(* IEC 61131-3 sources: AXOpen/src/showcase/app/src/components.kuka.robotics/Documentation, 7 files *)

(* ---- AxoKrc4_v_5_x_x_Krc5Showcase.st ---- *)
USING AXOpen.Core;

NAMESPACE AXOpen.Components.Kuka.Robotics
    {S7.extern=ReadWrite}
    CLASS AxoKrc4_v_5_x_x_Krc5Showcase EXTENDS AXOpen.Core.AxoObject
        //<ComponentDeclaration>
        VAR PUBLIC
            // KRC5 controller driven by the same AxoKrc4 proxy —
            // the slot-2 DIO512 layout is identical between KRC4 and KRC5.
            ExampleRobot : AXOpen.Components.Kuka.Robotics.v_5_x_x.AxoKrc4;
        END_VAR
        //</ComponentDeclaration>

        //<InitializationArgumentsDeclaration>
        VAR PUBLIC
            movementParams : AXOpen.Components.Abstractions.Robotics.AxoRoboticsMovementsParams;
            {#ix-set:AttributeName = "<#Activate manual control#>"}
            ActivateManualControl : BOOL;
        END_VAR
        //</InitializationArgumentsDeclaration>

        METHOD PUBLIC OVERRIDE Run
            VAR_INPUT
                inParent : IAxoObject;
            END_VAR

            SUPER.Run(inParent);

            IF ActivateManualControl THEN
                ExampleRobot.ActivateManualControl();
            END_IF;

            //<Initialization>
            // kuka_rb2_HwID points at the KRC5 device (192.168.100.106)
            // provisioned by the kuka_krc5_dio512 template in plc_line.hwl.yml.
            ExampleRobot.Run(THIS, AXOpen.Showcase.HwIdentifiers#kuka_rb2_HwID);
            //</Initialization>

            THIS.UseInSequencer();
        END_METHOD

        //<Usage>
        VAR PUBLIC
            Sequencer : AxoSequencer;
            Steps : ARRAY[0..19] OF AXOpen.Core.AxoStep;
        END_VAR

        METHOD PRIVATE UseInSequencer

            Sequencer.Run(THIS);
            Sequencer.Open();
            Sequencer.SequenceMode := eAxoSequenceMode#RunOnce;

            IF(Steps[0].Execute(Sequencer, 'Restore')) THEN
                ActivateManualControl := FALSE;
                ExampleRobot.Config.InfoTime      := LTIME#2S;
                ExampleRobot.Config.TaskTimeout   := LTIME#0S;
                ExampleRobot.Config.ErrorTime     := LTIME#0S;
                ExampleRobot.Restore();
                Sequencer.MoveNext();
            END_IF;

            IF(Steps[1].Execute(Sequencer, 'Start at main')) THEN
                IF(ExampleRobot.StartAtMain().IsDone()) THEN
                    Sequencer.MoveNext();
                END_IF;
            END_IF;

            IF(Steps[2].Execute(Sequencer, 'Start motors and program')) THEN
                IF(ExampleRobot.StartMotorsAndProgram().IsDone()) THEN
                    Sequencer.MoveNext();
                END_IF;
            END_IF;

            IF(Steps[3].Execute(Sequencer, 'Move to position 100')) THEN
                movementParams.ActionNo         :=  BYTE#100;
                movementParams.GlobalSpeed      :=  BYTE#5;
                movementParams.ToolNo           :=  BYTE#10;
                movementParams.WorkobjectNo     :=  BYTE#15;
                movementParams.PointNo          :=  BYTE#20;
                movementParams.UserSpecSpeed1   :=  INT#25;
                movementParams.UserSpecSpeed2   :=  INT#30;
                movementParams.Coordinates.X    :=  REAL#-1.2;
                movementParams.Coordinates.Y    :=  REAL#2.3;
                movementParams.Coordinates.Z    :=  REAL#3.4;
                movementParams.Coordinates.Rx   :=  REAL#4.5;
                movementParams.Coordinates.Ry   :=  REAL#5.6;
                movementParams.Coordinates.Rz   :=  REAL#6.7;

                IF(ExampleRobot.StartMovements(movementParams).IsDone()) THEN
                    ExampleRobot.StartMovementsTask.Restore();
                    Sequencer.MoveNext();
                END_IF;
            END_IF;

            IF(Steps[4].Execute(Sequencer, 'Move to position 1')) THEN
                movementParams.ActionNo             :=  BYTE#1;

                IF(ExampleRobot.StartMovements(movementParams).IsDone()) THEN
                    ExampleRobot.StartMovementsTask.Restore();
                    Sequencer.MoveNext();
                END_IF;
            END_IF;

            IF(Steps[5].Execute(Sequencer, 'Move to position 3')) THEN
                movementParams.ActionNo             :=  BYTE#3;

                IF(ExampleRobot.StartMovements(movementParams).IsBusy() AND Sequencer.CurrentStep.Duration >= T#500ms) THEN
                    Sequencer.MoveNext();
                END_IF;
            END_IF;

            IF(Steps[6].Execute(Sequencer, 'Stop during movement')) THEN
                ExampleRobot.StartMovements(movementParams);
                IF(ExampleRobot.StopMovements().IsDone()) THEN
                    Sequencer.MoveNext();
                END_IF;
            END_IF;

            IF(Steps[7].Execute(Sequencer, '<#Unlocking and opening the robotic cell#>')) THEN
                ExampleRobot.StartMovements(movementParams);
                IF (Sequencer.CurrentStep.Duration >= T#1s) THEN
                    Sequencer.MoveNext();
                END_IF;
            END_IF;

            IF (Steps[8].Execute(Sequencer, '<#Closing and locking the robotic cell#>')) THEN
                ExampleRobot.StartMovements(movementParams);
                IF (Sequencer.CurrentStep.Duration >= T#1s) THEN
                    Sequencer.MoveNext();
                END_IF;
            END_IF;

            IF(Steps[9].Execute(Sequencer, 'Start motors and program')) THEN
                ExampleRobot.StartMovements(movementParams);
                IF(ExampleRobot.StartMotorsAndProgram().IsDone() AND Sequencer.CurrentStep.Duration >= T#1s) THEN
                    Sequencer.MoveNext();
                END_IF;
            END_IF;

            IF(Steps[10].Execute(Sequencer, 'Continue to position 3')) THEN
                ExampleRobot.StartMovements(movementParams);
                IF(ExampleRobot.StartMovementsTask.IsDone()) THEN
                    ExampleRobot.StartMovementsTask.Restore();
                    Sequencer.MoveNext();
                END_IF;
            END_IF;

            IF(Steps[11].Execute(Sequencer, 'Move to position 100')) THEN
                movementParams.ActionNo             :=  BYTE#100;

                IF(ExampleRobot.StartMovements(movementParams).IsDone()) THEN
                    ExampleRobot.StartMovementsTask.Restore();
                    Sequencer.MoveNext();
                END_IF;
            END_IF;

            IF(Steps[12].Execute(Sequencer, 'Move to position 1')) THEN
                movementParams.ActionNo             :=  BYTE#1;

                IF(ExampleRobot.StartMovements(movementParams).IsDone()) THEN
                    ExampleRobot.StartMovementsTask.Restore();
                    Sequencer.MoveNext();
                END_IF;
            END_IF;

            IF(Steps[13].Execute(Sequencer, 'Stop movement and program')) THEN
                IF(ExampleRobot.StopMovementsAndProgram().IsDone()) THEN
                    Sequencer.MoveNext();
                END_IF;
            END_IF;

            IF(Steps[14].Execute(Sequencer, 'Stop motors')) THEN
                IF(ExampleRobot.StopMotors().IsDone()) THEN
                    Sequencer.MoveNext();
                END_IF;
            END_IF;

            IF(Steps[15].Execute(Sequencer, 'Reset all outputs')) THEN
                IF(ExampleRobot.ResetAllOutputs().IsDone()) THEN
                    Sequencer.MoveNext();
                END_IF;
            END_IF;

            IF(Steps[16].Execute(Sequencer, 'Start motors, program and movements combined')) THEN
                IF(ExampleRobot.StartMotorsProgramAndMovements(movementParams).IsDone()) THEN
                    Sequencer.MoveNext();
                END_IF;
            END_IF;

            IF(Steps[17].Execute(Sequencer, 'Stop program')) THEN
                IF(ExampleRobot.StopProgram().IsDone()) THEN
                    Sequencer.MoveNext();
                END_IF;
            END_IF;

            IF(Steps[18].Execute(Sequencer, 'Start program')) THEN
                IF(ExampleRobot.StartProgram().IsDone()) THEN
                    Sequencer.MoveNext();
                END_IF;
            END_IF;

            IF(Steps[19].Execute(Sequencer, 'Restore')) THEN
                ExampleRobot.Restore();
                Sequencer.CompleteSequence();
            END_IF;
        END_METHOD

        //</Usage>
    END_CLASS
END_NAMESPACE

(* ---- AxoKrc4_v_5_x_x_ManualControl.st ---- *)
USING AXOpen.Core;
USING AXOpen.Components.Abstractions.Robotics;

NAMESPACE AXOpen.Components.Kuka.Robotics.v_5_x_x
    {S7.extern=ReadWrite}
    CLASS AxoKrc4_v_5_x_x_ManualControl EXTENDS AXOpen.Core.AxoObject
        //<ComponentDeclaration>
        VAR PUBLIC
            ManualRobot : AXOpen.Components.Kuka.Robotics.v_5_x_x.AxoKrc4;
        END_VAR
        //</ComponentDeclaration>

        //<InitializationArgumentsDeclaration>
        VAR PUBLIC
            manualMovementParams : AXOpen.Components.Abstractions.Robotics.AxoRoboticsMovementsParams;
            {#ix-set:AttributeName = "<#Engage manual control#>"}
            EngageManualControl : BOOL;
            {#ix-set:AttributeName = "<#Trigger manual move (one shot)#>"}
            TriggerManualMove : BOOL;
        END_VAR
        //</InitializationArgumentsDeclaration>

        METHOD PUBLIC OVERRIDE Run
            VAR_INPUT
                inParent : IAxoObject;
            END_VAR

            SUPER.Run(inParent);

            ManualRobot.Config.InfoTime    := LTIME#2S;
            ManualRobot.Config.ErrorTime   := LTIME#0S;
            ManualRobot.Config.TaskTimeout := LTIME#0S;

            //<Initialization>
            ManualRobot.Run(inParent := THIS,
                            hwID     := AXOpen.Showcase.HwIdentifiers#kuka_rb1_HwID);
            //</Initialization>

            //<ManualControlActivation>
            // ActivateManualControl() must be called every cycle while the
            // operator drives the component from the HMI. The component
            // bypasses the automatic task pipeline and exposes raw command
            // signals through its dedicated views.
            IF EngageManualControl THEN
                ManualRobot.ActivateManualControl();
            END_IF;
            //</ManualControlActivation>

            //<ManualMoveTrigger>
            // The HMI can pre-load movement parameters and fire a single
            // StartMovements() invocation. When the task completes the
            // operator restores it from its terminal state to be ready
            // for the next manual command.
            IF TriggerManualMove THEN
                manualMovementParams.ActionNo       :=  BYTE#1;
                manualMovementParams.GlobalSpeed    :=  BYTE#10;
                manualMovementParams.ToolNo         :=  BYTE#1;
                manualMovementParams.WorkobjectNo   :=  BYTE#1;
                manualMovementParams.PointNo        :=  BYTE#1;
                IF ManualRobot.StartMovements(manualMovementParams).IsDone() THEN
                    ManualRobot.StartMovementsTask.Restore();
                    TriggerManualMove := FALSE;
                END_IF;
            END_IF;
            //</ManualMoveTrigger>
        END_METHOD
    END_CLASS
END_NAMESPACE

(* ---- AxoKrc4_v_5_x_x_Showcase.st ---- *)
USING AXOpen.Core;
USING AXOpen.Components.Abstractions.Robotics;

NAMESPACE AXOpen.Components.Kuka.Robotics.v_5_x_x
    {S7.extern=ReadWrite}
    CLASS AxoKrc4_v_5_x_x_Showcase EXTENDS AXOpen.Core.AxoObject
        //<ComponentDeclaration>
        VAR PUBLIC
            ExampleRobot : AXOpen.Components.Kuka.Robotics.v_5_x_x.AxoKrc4;
        END_VAR
        //</ComponentDeclaration>

        //<InitializationArgumentsDeclaration>
        VAR PUBLIC
            movementParams : AXOpen.Components.Abstractions.Robotics.AxoRoboticsMovementsParams;
            {#ix-set:AttributeName = "<#Activate manual control#>"}
            ActivateManualControl : BOOL;
        END_VAR
        //</InitializationArgumentsDeclaration>

        METHOD PUBLIC OVERRIDE Run
            VAR_INPUT
                inParent : IAxoObject;
            END_VAR

            SUPER.Run(inParent);

            IF ActivateManualControl THEN
                ExampleRobot.ActivateManualControl();
            END_IF;

            ExampleRobot.Config.ErrorTime := T#0s;
            //<Initialization>
            ExampleRobot.Run(THIS,AXOpen.Showcase.HwIdentifiers#kuka_rb1_HwID);
            //</Initialization>

        THIS.UseInSequencer();
        END_METHOD

        //<Usage>
        VAR PUBLIC
            Sequencer : AxoSequencer;
            Steps : ARRAY[0..19] OF AXOpen.Core.AxoStep;
        END_VAR

        METHOD PRIVATE UseInSequencer

            Sequencer.Run(THIS);
            Sequencer.Open();
            Sequencer.SequenceMode := eAxoSequenceMode#RunOnce;

            IF(Steps[0].Execute(Sequencer, 'Restore')) THEN
                ActivateManualControl := FALSE;
                ExampleRobot.Config.InfoTime      := LTIME#2S;
                ExampleRobot.Config.TaskTimeout   := LTIME#0S;
                ExampleRobot.Config.ErrorTime     := LTIME#0S;
                ExampleRobot.Restore();
                Sequencer.MoveNext();
            END_IF;

            IF(Steps[1].Execute(Sequencer, 'Start at main')) THEN
                IF(ExampleRobot.StartAtMain().IsDone()) THEN
                    Sequencer.MoveNext();
                END_IF;
            END_IF;

            IF(Steps[2].Execute(Sequencer, 'Start motors and program')) THEN
                IF(ExampleRobot.StartMotorsAndProgram().IsDone()) THEN
                    Sequencer.MoveNext();
                END_IF;
            END_IF;

            IF(Steps[3].Execute(Sequencer, 'Move to position 100')) THEN
                movementParams.ActionNo         :=  BYTE#100;
                movementParams.GlobalSpeed      :=  BYTE#5;
                movementParams.ToolNo           :=  BYTE#10;
                movementParams.WorkobjectNo     :=  BYTE#15;
                movementParams.PointNo          :=  BYTE#20;
                movementParams.UserSpecSpeed1   :=  INT#25;
                movementParams.UserSpecSpeed2   :=  INT#30;
                movementParams.Coordinates.X    :=  REAL#-1.2;
                movementParams.Coordinates.Y    :=  REAL#2.3;
                movementParams.Coordinates.Z    :=  REAL#3.4;
                movementParams.Coordinates.Rx   :=  REAL#4.5;
                movementParams.Coordinates.Ry   :=  REAL#5.6;
                movementParams.Coordinates.Rz   :=  REAL#6.7;

                IF(ExampleRobot.StartMovements(movementParams).IsDone()) THEN
                    ExampleRobot.StartMovementsTask.Restore();
                    Sequencer.MoveNext();
                END_IF;
            END_IF;

            IF(Steps[4].Execute(Sequencer, 'Move to position 1')) THEN
                movementParams.ActionNo             :=  BYTE#1;

                IF(ExampleRobot.StartMovements(movementParams).IsDone()) THEN
                    ExampleRobot.StartMovementsTask.Restore();
                    Sequencer.MoveNext();
                END_IF;
            END_IF;

            IF(Steps[5].Execute(Sequencer, 'Move to position 3')) THEN
                movementParams.ActionNo             :=  BYTE#3;

                IF(ExampleRobot.StartMovements(movementParams).IsBusy() AND Sequencer.CurrentStep.Duration >= T#500ms) THEN
                    Sequencer.MoveNext();
                END_IF;
            END_IF;
            // Simulation of the entering the robotic cell during movement =>
            IF(Steps[6].Execute(Sequencer, 'Stop during movement')) THEN
                ExampleRobot.StartMovements(movementParams); // <- This line just emulates the cyclical call of the movement method
                IF(ExampleRobot.StopMovements(eAxoRoboticsStopType#Soft).IsDone()) THEN
                    Sequencer.MoveNext();
                END_IF;
            END_IF;

            IF(Steps[7].Execute(Sequencer, '<#Unlocking and opening the robotic cell#>')) THEN
                //-------------------------------------------------------
                ExampleRobot.StartMovements(movementParams); // <- This line just emulates the cyclical call of the movement method
                IF (Sequencer.CurrentStep.Duration >= T#1s) THEN    // IF (TRUE) THEN
                    Sequencer.MoveNext();
                END_IF;
                //-------------------------------------------------------
            END_IF;

            IF (Steps[8].Execute(Sequencer, '<#Closing and locking the robotic cell#>')) THEN
                //-------------------------------------------------------
                ExampleRobot.StartMovements(movementParams); // <- This line just emulates the cyclical call of the movement method
                IF (Sequencer.CurrentStep.Duration >= T#1s) THEN    // IF (TRUE) THEN
                    Sequencer.MoveNext();
                END_IF;
                //-------------------------------------------------------
            END_IF;
            // <= Simulation of the entering the robotic cell during movement

            IF(Steps[9].Execute(Sequencer, 'Start motors and program')) THEN
                ExampleRobot.StartMovements(movementParams); // <- This line just emulates the cyclical call of the movement method
                IF(ExampleRobot.StartMotorsAndProgram().IsDone() AND Sequencer.CurrentStep.Duration >= T#1s) THEN //IF(ExampleRobot.StartMotorsAndProgram().IsDone()) THEN // <- Starting motor and program after safety circuit has been interupted
                    Sequencer.MoveNext();
                END_IF;
            END_IF;

            IF(Steps[10].Execute(Sequencer, 'Continue to position 3')) THEN
                ExampleRobot.StartMovements(movementParams); // <- This line just emulates the cyclical call of the movement method
                IF(ExampleRobot.StartMovementsTask.IsDone()) THEN
                    ExampleRobot.StartMovementsTask.Restore();
                    Sequencer.MoveNext();
                END_IF;
            END_IF;

            IF(Steps[11].Execute(Sequencer, 'Move to position 100')) THEN
                movementParams.ActionNo             :=  BYTE#100;

                IF(ExampleRobot.StartMovements(movementParams).IsDone()) THEN
                    ExampleRobot.StartMovementsTask.Restore();
                    Sequencer.MoveNext();
                END_IF;
            END_IF;

            IF(Steps[12].Execute(Sequencer, 'Move to position 1')) THEN
                movementParams.ActionNo             :=  BYTE#1;

                IF(ExampleRobot.StartMovements(movementParams).IsDone()) THEN
                    ExampleRobot.StartMovementsTask.Restore();
                    Sequencer.MoveNext();
                END_IF;
            END_IF;

            IF(Steps[13].Execute(Sequencer, 'Stop movement and program')) THEN
                IF(ExampleRobot.StopMovementsAndProgram(eAxoRoboticsStopType#Soft).IsDone()) THEN
                    Sequencer.MoveNext();
                END_IF;
            END_IF;

            IF(Steps[14].Execute(Sequencer, 'Stop motors')) THEN
                IF(ExampleRobot.StopMotors().IsDone()) THEN
                    Sequencer.MoveNext();
                END_IF;
            END_IF;

            IF(Steps[15].Execute(Sequencer, 'Reset all outputs')) THEN
                IF(ExampleRobot.ResetAllOutputs().IsDone()) THEN
                    Sequencer.MoveNext();
                END_IF;
            END_IF;

            IF(Steps[16].Execute(Sequencer, 'Start motors, program and movements combined')) THEN
                IF(ExampleRobot.StartMotorsProgramAndMovements(movementParams).IsDone()) THEN
                    Sequencer.MoveNext();
                END_IF;
            END_IF;

            IF(Steps[17].Execute(Sequencer, 'Stop program')) THEN
                IF(ExampleRobot.StopProgram().IsDone()) THEN
                    Sequencer.MoveNext();
                END_IF;
            END_IF;

            IF(Steps[18].Execute(Sequencer, 'Start program')) THEN
                IF(ExampleRobot.StartProgram().IsDone()) THEN
                    Sequencer.MoveNext();
                END_IF;
            END_IF;

            IF(Steps[19].Execute(Sequencer, 'Restore')) THEN
                ExampleRobot.Restore();
                Sequencer.CompleteSequence();
            END_IF;
        END_METHOD

        //</Usage>
    END_CLASS
END_NAMESPACE

(* ---- AxoKrc4_v_5_x_x_Showcase2.st ---- *)
USING AXOpen.Core;

NAMESPACE AXOpen.Components.Kuka.Robotics
    {S7.extern=ReadWrite}
    CLASS AxoKrc4_v_5_x_x_Showcase2 EXTENDS AXOpen.Core.AxoObject
        //<ComponentDeclaration>
        VAR PUBLIC
            ExampleRobot : AXOpen.Components.Kuka.Robotics.v_5_x_x.AxoKrc4;
        END_VAR
        //</ComponentDeclaration>

        //<InitializationArgumentsDeclaration>
        VAR PUBLIC
            movementParams : AXOpen.Components.Abstractions.Robotics.AxoRoboticsMovementsParams;
            {#ix-set:AttributeName = "<#Activate manual control#>"}
            ActivateManualControl : BOOL;
        END_VAR
        //</InitializationArgumentsDeclaration>

        METHOD PUBLIC OVERRIDE Run
            VAR_INPUT
                inParent : IAxoObject;
            END_VAR

            SUPER.Run(inParent);

            IF ActivateManualControl THEN
                ExampleRobot.ActivateManualControl();
            END_IF;

            //<Initialization>
            ExampleRobot.Run(THIS,AXOpen.Showcase.HwIdentifiers#kuka_rb1_HwID);
            //</Initialization>

            THIS.UseInSequencer();
        END_METHOD

        //<Usage>
        VAR PUBLIC
            Sequencer : AxoSequencer;
            Steps : ARRAY[0..14] OF AXOpen.Core.AxoStep;
        END_VAR

        METHOD PRIVATE UseInSequencer

            Sequencer.Run(THIS);
            Sequencer.Open();
            Sequencer.SequenceMode := eAxoSequenceMode#RunOnce;

            IF(Steps[0].Execute(Sequencer, 'Restore')) THEN
                ActivateManualControl := FALSE;
                ExampleRobot.Config.TaskTimeout   := LTIME#0S;
                ExampleRobot.Config.ErrorTime     := LTIME#0S;
                ExampleRobot.Restore();
                Sequencer.MoveNext();
            END_IF;

            IF(Steps[1].Execute(Sequencer, 'Start at main')) THEN
                IF(ExampleRobot.StartAtMain().IsDone()) THEN
                    Sequencer.MoveNext();
                END_IF;
            END_IF;

            IF(Steps[2].Execute(Sequencer, 'Start motors and program')) THEN
                IF(ExampleRobot.StartMotorsAndProgram().IsDone()) THEN
                    Sequencer.MoveNext();
                END_IF;
            END_IF;

            IF(Steps[3].Execute(Sequencer, 'Move to position 100')) THEN
                movementParams.ActionNo         :=  BYTE#100;
                movementParams.GlobalSpeed      :=  BYTE#5;
                movementParams.ToolNo           :=  BYTE#10;
                movementParams.WorkobjectNo     :=  BYTE#15;
                movementParams.PointNo          :=  BYTE#20;
                movementParams.UserSpecSpeed1   :=  INT#25;
                movementParams.UserSpecSpeed2   :=  INT#30;
                movementParams.Coordinates.X    :=  REAL#-1.2;
                movementParams.Coordinates.Y    :=  REAL#2.3;
                movementParams.Coordinates.Z    :=  REAL#3.4;
                movementParams.Coordinates.Rx   :=  REAL#4.5;
                movementParams.Coordinates.Ry   :=  REAL#5.6;
                movementParams.Coordinates.Rz   :=  REAL#6.7;

                IF(ExampleRobot.StartMovements(movementParams).IsDone()) THEN
                    ExampleRobot.StartMovementsTask.Restore();
                    Sequencer.MoveNext();
                END_IF;
            END_IF;

            IF(Steps[4].Execute(Sequencer, 'Move to position 1')) THEN
                movementParams.ActionNo             :=  BYTE#1;

                IF(ExampleRobot.StartMovements(movementParams).IsDone()) THEN
                    ExampleRobot.StartMovementsTask.Restore();
                    Sequencer.MoveNext();
                END_IF;
            END_IF;

            IF(Steps[5].Execute(Sequencer, 'Move to position 3')) THEN
                movementParams.ActionNo             :=  BYTE#3;

                IF(ExampleRobot.StartMovements(movementParams).IsBusy() AND Sequencer.CurrentStep.Duration >= T#500ms) THEN
                    Sequencer.MoveNext();
                END_IF;
            END_IF;
            // Simulation of the entering the robotic cell during movement =>
            IF(Steps[6].Execute(Sequencer, 'Stop during movement')) THEN
                ExampleRobot.StartMovements(movementParams); // <- This line just emulates the cyclical call of the movement method
                IF(ExampleRobot.StopMovements().IsDone()) THEN
                    Sequencer.MoveNext();
                END_IF;
            END_IF;

            IF(Steps[7].Execute(Sequencer, '<#Unlocking and opening the robotic cell#>')) THEN
                //-------------------------------------------------------
                ExampleRobot.StartMovements(movementParams); // <- This line just emulates the cyclical call of the movement method
                IF (Sequencer.CurrentStep.Duration >= T#1s) THEN    // IF (TRUE) THEN
                    Sequencer.MoveNext();
                END_IF;
                //-------------------------------------------------------
            END_IF;

            IF (Steps[8].Execute(Sequencer, '<#Closing and locking the robotic cell#>')) THEN
                //-------------------------------------------------------
                ExampleRobot.StartMovements(movementParams); // <- This line just emulates the cyclical call of the movement method
                IF (Sequencer.CurrentStep.Duration >= T#1s) THEN    // IF (TRUE) THEN
                    Sequencer.MoveNext();
                END_IF;
                //-------------------------------------------------------
            END_IF;
            // <= Simulation of the entering the robotic cell during movement

            IF(Steps[9].Execute(Sequencer, 'Start motors and program')) THEN
                ExampleRobot.StartMovements(movementParams); // <- This line just emulates the cyclical call of the movement method
                IF(ExampleRobot.StartMotorsAndProgram().IsDone() AND Sequencer.CurrentStep.Duration >= T#1s) THEN //IF(ExampleRobot.StartMotorsAndProgram().IsDone()) THEN // <- Starting motor and program after safety circuit has been interupted
                    Sequencer.MoveNext();
                END_IF;
            END_IF;

            IF(Steps[10].Execute(Sequencer, 'Continue to position 3')) THEN
                ExampleRobot.StartMovements(movementParams); // <- This line just emulates the cyclical call of the movement method
                IF(ExampleRobot.StartMovementsTask.IsDone()) THEN
                    ExampleRobot.StartMovementsTask.Restore();
                    Sequencer.MoveNext();
                END_IF;
            END_IF;

            IF(Steps[11].Execute(Sequencer, 'Move to position 100')) THEN
                movementParams.ActionNo             :=  BYTE#100;

                IF(ExampleRobot.StartMovements(movementParams).IsDone()) THEN
                    ExampleRobot.StartMovementsTask.Restore();
                    Sequencer.MoveNext();
                END_IF;
            END_IF;

            IF(Steps[12].Execute(Sequencer, 'Move to position 1')) THEN
                movementParams.ActionNo             :=  BYTE#1;

                IF(ExampleRobot.StartMovements(movementParams).IsDone()) THEN
                    ExampleRobot.StartMovementsTask.Restore();
                    Sequencer.MoveNext();
                END_IF;
            END_IF;

            IF(Steps[13].Execute(Sequencer, 'Stop movement and program')) THEN
                IF(ExampleRobot.StopMovementsAndProgram().IsDone()) THEN
                    Sequencer.MoveNext();
                END_IF;
            END_IF;
            IF(Steps[14].Execute(Sequencer, 'Restore')) THEN
                ExampleRobot.Restore();
                Sequencer.CompleteSequence();
            END_IF;
        END_METHOD

        //</Usage>
    END_CLASS
END_NAMESPACE

(* ---- AxoKrc5_v_5_x_x_ManualControl.st ---- *)
USING AXOpen.Core;
USING AXOpen.Components.Abstractions.Robotics;

NAMESPACE AXOpen.Components.Kuka.Robotics.v_5_x_x
    {S7.extern=ReadWrite}
    CLASS AxoKrc5_v_5_x_x_ManualControl EXTENDS AXOpen.Core.AxoObject
        //<ComponentDeclaration>
        VAR PUBLIC
            ManualRobot : AXOpen.Components.Kuka.Robotics.v_5_x_x.AxoKrc5;
        END_VAR
        //</ComponentDeclaration>

        //<InitializationArgumentsDeclaration>
        VAR PUBLIC
            manualMovementParams : AXOpen.Components.Abstractions.Robotics.AxoRoboticsMovementsParams;
            {#ix-set:AttributeName = "<#Engage manual control#>"}
            EngageManualControl : BOOL;
            {#ix-set:AttributeName = "<#Trigger manual move (one shot)#>"}
            TriggerManualMove : BOOL;
        END_VAR
        //</InitializationArgumentsDeclaration>

        METHOD PUBLIC OVERRIDE Run
            VAR_INPUT
                inParent : IAxoObject;
            END_VAR

            SUPER.Run(inParent);

            ManualRobot.Config.InfoTime    := LTIME#2S;
            ManualRobot.Config.ErrorTime   := LTIME#0S;
            ManualRobot.Config.TaskTimeout := LTIME#0S;

            //<Initialization>
            ManualRobot.Run(inParent := THIS,
                            hwID     := AXOpen.Showcase.HwIdentifiers#kuka_rb2_HwID);
            //</Initialization>

            //<ManualControlActivation>
            // ActivateManualControl() must be called every cycle while the
            // operator drives the component from the HMI. The component
            // bypasses the automatic task pipeline and exposes raw command
            // signals through its dedicated views.
            IF EngageManualControl THEN
                ManualRobot.ActivateManualControl();
            END_IF;
            //</ManualControlActivation>

            //<ManualMoveTrigger>
            // The HMI can pre-load movement parameters and fire a single
            // StartMovements() invocation. When the task completes the
            // operator restores it from its terminal state to be ready
            // for the next manual command.
            IF TriggerManualMove THEN
                manualMovementParams.ActionNo       :=  BYTE#1;
                manualMovementParams.GlobalSpeed    :=  BYTE#10;
                manualMovementParams.ToolNo         :=  BYTE#1;
                manualMovementParams.WorkobjectNo   :=  BYTE#1;
                manualMovementParams.PointNo        :=  BYTE#1;
                IF ManualRobot.StartMovements(manualMovementParams).IsDone() THEN
                    ManualRobot.StartMovementsTask.Restore();
                    TriggerManualMove := FALSE;
                END_IF;
            END_IF;
            //</ManualMoveTrigger>
        END_METHOD
    END_CLASS
END_NAMESPACE

(* ---- AxoKrc5_v_5_x_x_Showcase.st ---- *)
USING AXOpen.Core;
USING AXOpen.Components.Abstractions.Robotics;

NAMESPACE AXOpen.Components.Kuka.Robotics.v_5_x_x
    {S7.extern=ReadWrite}
    CLASS AxoKrc5_v_5_x_x_Showcase EXTENDS AXOpen.Core.AxoObject
        //<ComponentDeclaration>
        VAR PUBLIC
            ExampleRobot : AXOpen.Components.Kuka.Robotics.v_5_x_x.AxoKrc5;
        END_VAR
        //</ComponentDeclaration>

        //<InitializationArgumentsDeclaration>
        VAR PUBLIC
            movementParams : AXOpen.Components.Abstractions.Robotics.AxoRoboticsMovementsParams;
            {#ix-set:AttributeName = "<#Activate manual control#>"}
            ActivateManualControl : BOOL;
        END_VAR
        //</InitializationArgumentsDeclaration>

        METHOD PUBLIC OVERRIDE Run
            VAR_INPUT
                inParent : IAxoObject;
            END_VAR

            SUPER.Run(inParent);

            IF ActivateManualControl THEN
                ExampleRobot.ActivateManualControl();
            END_IF;

            //<Initialization>
            ExampleRobot.Run(THIS,AXOpen.Showcase.HwIdentifiers#kuka_rb2_HwID);
            //</Initialization>

            THIS.UseInSequencer();
        END_METHOD

        //<Usage>
        VAR PUBLIC
            Sequencer : AxoSequencer;
            Steps : ARRAY[0..20] OF AXOpen.Core.AxoStep;
            {#ix-set:AttributeName = "<#Last byte received from robot#>"}
            _lastByteFromRobot : BYTE;
        END_VAR

        METHOD PRIVATE UseInSequencer

            Sequencer.Run(THIS);
            Sequencer.Open();
            Sequencer.SequenceMode := eAxoSequenceMode#RunOnce;

            IF(Steps[0].Execute(Sequencer, 'Restore')) THEN
                ActivateManualControl := FALSE;
                ExampleRobot.Config.InfoTime      := LTIME#2S;
                ExampleRobot.Config.TaskTimeout   := LTIME#0S;
                ExampleRobot.Config.ErrorTime     := LTIME#0S;
                ExampleRobot.Restore();
                Sequencer.MoveNext();
            END_IF;

            IF(Steps[1].Execute(Sequencer, 'Start at main')) THEN
                IF(ExampleRobot.StartAtMain().IsDone()) THEN
                    Sequencer.MoveNext();
                END_IF;
            END_IF;

            IF(Steps[2].Execute(Sequencer, 'Start motors and program')) THEN
                IF(ExampleRobot.StartMotorsAndProgram().IsDone()) THEN
                    Sequencer.MoveNext();
                END_IF;
            END_IF;

            IF(Steps[3].Execute(Sequencer, 'Move to position 100')) THEN
                movementParams.ActionNo         :=  BYTE#100;
                movementParams.GlobalSpeed      :=  BYTE#5;
                movementParams.ToolNo           :=  BYTE#10;
                movementParams.WorkobjectNo     :=  BYTE#15;
                movementParams.PointNo          :=  BYTE#20;
                movementParams.UserSpecSpeed1   :=  INT#25;
                movementParams.UserSpecSpeed2   :=  INT#30;
                movementParams.Coordinates.X    :=  REAL#-1.2;
                movementParams.Coordinates.Y    :=  REAL#2.3;
                movementParams.Coordinates.Z    :=  REAL#3.4;
                movementParams.Coordinates.Rx   :=  REAL#4.5;
                movementParams.Coordinates.Ry   :=  REAL#5.6;
                movementParams.Coordinates.Rz   :=  REAL#6.7;

                IF(ExampleRobot.StartMovements(movementParams).IsDone()) THEN
                    ExampleRobot.StartMovementsTask.Restore();
                    Sequencer.MoveNext();
                END_IF;
            END_IF;

            IF(Steps[4].Execute(Sequencer, 'Move to position 1')) THEN
                movementParams.ActionNo             :=  BYTE#1;

                IF(ExampleRobot.StartMovements(movementParams).IsDone()) THEN
                    ExampleRobot.StartMovementsTask.Restore();
                    Sequencer.MoveNext();
                END_IF;
            END_IF;

            IF(Steps[5].Execute(Sequencer, 'Move to position 3')) THEN
                movementParams.ActionNo             :=  BYTE#3;

                IF(ExampleRobot.StartMovements(movementParams).IsBusy() AND Sequencer.CurrentStep.Duration >= T#500ms) THEN
                    Sequencer.MoveNext();
                END_IF;
            END_IF;
            // Simulation of the entering the robotic cell during movement =>
            IF(Steps[6].Execute(Sequencer, 'Stop during movement')) THEN
                ExampleRobot.StartMovements(movementParams); // <- This line just emulates the cyclical call of the movement method
                IF(ExampleRobot.StopMovements(eAxoRoboticsStopType#Soft).IsDone()) THEN
                    Sequencer.MoveNext();
                END_IF;
            END_IF;

            IF(Steps[7].Execute(Sequencer, '<#Unlocking and opening the robotic cell#>')) THEN
                //-------------------------------------------------------
                ExampleRobot.StartMovements(movementParams); // <- This line just emulates the cyclical call of the movement method
                IF (Sequencer.CurrentStep.Duration >= T#1s) THEN    // IF (TRUE) THEN
                    Sequencer.MoveNext();
                END_IF;
                //-------------------------------------------------------
            END_IF;

            IF (Steps[8].Execute(Sequencer, '<#Closing and locking the robotic cell#>')) THEN
                //-------------------------------------------------------
                ExampleRobot.StartMovements(movementParams); // <- This line just emulates the cyclical call of the movement method
                IF (Sequencer.CurrentStep.Duration >= T#1s) THEN    // IF (TRUE) THEN
                    Sequencer.MoveNext();
                END_IF;
                //-------------------------------------------------------
            END_IF;
            // <= Simulation of the entering the robotic cell during movement

            IF(Steps[9].Execute(Sequencer, 'Start motors and program')) THEN
                ExampleRobot.StartMovements(movementParams); // <- This line just emulates the cyclical call of the movement method
                IF(ExampleRobot.StartMotorsAndProgram().IsDone() AND Sequencer.CurrentStep.Duration >= T#1s) THEN //IF(ExampleRobot.StartMotorsAndProgram().IsDone()) THEN // <- Starting motor and program after safety circuit has been interupted
                    Sequencer.MoveNext();
                END_IF;
            END_IF;

            IF(Steps[10].Execute(Sequencer, 'Continue to position 3')) THEN
                ExampleRobot.StartMovements(movementParams); // <- This line just emulates the cyclical call of the movement method
                IF(ExampleRobot.StartMovementsTask.IsDone()) THEN
                    ExampleRobot.StartMovementsTask.Restore();
                    Sequencer.MoveNext();
                END_IF;
            END_IF;

            IF(Steps[11].Execute(Sequencer, 'Move to position 100')) THEN
                movementParams.ActionNo             :=  BYTE#100;

                IF(ExampleRobot.StartMovements(movementParams).IsDone()) THEN
                    ExampleRobot.StartMovementsTask.Restore();
                    Sequencer.MoveNext();
                END_IF;
            END_IF;

            IF(Steps[12].Execute(Sequencer, 'Move to position 1')) THEN
                movementParams.ActionNo             :=  BYTE#1;

                IF(ExampleRobot.StartMovements(movementParams).IsDone()) THEN
                    ExampleRobot.StartMovementsTask.Restore();
                    Sequencer.MoveNext();
                END_IF;
            END_IF;

            IF(Steps[13].Execute(Sequencer, 'Stop movement and program')) THEN
                IF(ExampleRobot.StopMovementsAndProgram(eAxoRoboticsStopType#Soft).IsDone()) THEN
                    Sequencer.MoveNext();
                END_IF;
            END_IF;

            IF(Steps[14].Execute(Sequencer, 'Stop motors')) THEN
                IF(ExampleRobot.StopMotors().IsDone()) THEN
                    Sequencer.MoveNext();
                END_IF;
            END_IF;

            IF(Steps[15].Execute(Sequencer, 'Reset all outputs')) THEN
                IF(ExampleRobot.ResetAllOutputs().IsDone()) THEN
                    Sequencer.MoveNext();
                END_IF;
            END_IF;

            IF(Steps[16].Execute(Sequencer, 'Start motors, program and movements combined')) THEN
                IF(ExampleRobot.StartMotorsProgramAndMovements(movementParams).IsDone()) THEN
                    Sequencer.MoveNext();
                END_IF;
            END_IF;

            IF(Steps[17].Execute(Sequencer, 'Stop program')) THEN
                IF(ExampleRobot.StopProgram().IsDone()) THEN
                    Sequencer.MoveNext();
                END_IF;
            END_IF;

            IF(Steps[18].Execute(Sequencer, 'Start program')) THEN
                IF(ExampleRobot.StartProgram().IsDone()) THEN
                    Sequencer.MoveNext();
                END_IF;
            END_IF;

            //<DataExchange>
            // KRC5-only raw passthrough (#1148): the component transports these
            // byte arrays verbatim over the same 64-byte cyclic block, without
            // interpreting them. They carry `RenderIgnore`, so they are not part
            // of the proxy view — exchange them from application code instead.
            IF(Steps[19].Execute(Sequencer, '<#Exchange raw data with the robot#>')) THEN
                // PLC -> robot: write an application-defined payload
                // (mapped onto output bytes 44..63 of the cyclic block).
                ExampleRobot.DataFromPlcToRobot[0]  := BYTE#16#A1;
                ExampleRobot.DataFromPlcToRobot[1]  := BYTE#16#B2;
                ExampleRobot.DataFromPlcToRobot[19] := BYTE#16#FF;

                // robot -> PLC: read the bytes the robot publishes back
                // (mapped from input bytes 48..63 of the cyclic block).
                _lastByteFromRobot := ExampleRobot.DataFromRobotToPlc[0];

                IF(Sequencer.CurrentStep.Duration >= T#500ms) THEN
                    Sequencer.MoveNext();
                END_IF;
            END_IF;
            //</DataExchange>

            IF(Steps[20].Execute(Sequencer, 'Restore')) THEN
                ExampleRobot.Restore();
                Sequencer.CompleteSequence();
            END_IF;
        END_METHOD

        //</Usage>
    END_CLASS
END_NAMESPACE

(* ---- KukaRobotics.st ---- *)
USING AXOpen.Components.Kuka.Robotics.v_5_x_x;

NAMESPACE AXOpen.Components.Kuka.Robotics
    {S7.extern=ReadWrite}
    CLASS KukaRobotics EXTENDS AXOpen.Core.AxoObject
        VAR PUBLIC
            _rootObject : AxoObject;
            axoKrc4_v_5_x_x         : AxoKrc4_v_5_x_x_Showcase;
            axoKrc5_v_5_x_x         : AxoKrc5_v_5_x_x_Showcase;
        END_VAR

        METHOD PUBLIC Execute
            _rootObject.Run(THIS);
            axoKrc4_v_5_x_x.Run(_rootObject);
            axoKrc5_v_5_x_x.Run(_rootObject);
        END_METHOD
    END_CLASS
END_NAMESPACE
